DATA_BLOCK "ST10_DeviceError"
{ S7_Optimized_Access := 'FALSE' }
VERSION : 0.1
   STRUCT
      CylinderFault : Struct
         C1GoWorkFault : Bool;
         C1GoHomeFault : Bool;
         C1SensorPositionFault : Bool;
         C1SpareFault : Bool;
         C2GoWorkFault : Bool;
         C2GoHomeFault : Bool;
         C2SensorPositionFault : Bool;
         C2SpareFault : Bool;
         C3GoWorkFault : Bool;
         C3GoHomeFault : Bool;
         C3SensorPositionFault : Bool;
         C3SpareFault : Bool;
         C4GoWorkFault : Bool;
         C4GoHomeFault : Bool;
         C4SensorPositionFault : Bool;
         C4SpareFault : Bool;
         C5GoWorkFault : Bool;
         C5GoHomeFault : Bool;
         C5SensorPositionFault : Bool;
         C5SpareFault : Bool;
         C6GoWorkFault : Bool;
         C6GoHomeFault : Bool;
         C6SensorPositionFault : Bool;
         C6SpareFault : Bool;
         C7GoWorkFault : Bool;
         C7GoHomeFault : Bool;
         C7SensorPositionFault : Bool;
         C7SpareFault : Bool;
         C8GoWorkFault : Bool;
         C8GoHomeFault : Bool;
         C8SensorPositionFault : Bool;
         C8SpareFault : Bool;
         C9GoWorkFault : Bool;
         C9GoHomeFault : Bool;
         C9SensorPositionFault : Bool;
         C9SpareFault : Bool;
         C10GoWorkFault : Bool;
         C10GoHomeFault : Bool;
         C10SensorPositionFault : Bool;
         C10SpareFault : Bool;
         C11GoWorkFault : Bool;
         C11GoHomeFault : Bool;
         C11SensorPositionFault : Bool;
         C11SpareFault : Bool;
         C12GoWorkFault : Bool;
         C12GoHomeFault : Bool;
         C12SensorPositionFault : Bool;
         C12SpareFault : Bool;
         C13GoWorkFault : Bool;
         C13GoHomeFault : Bool;
         C13SensorPositionFault : Bool;
         C13SpareFault : Bool;
         C14GoWorkFault : Bool;
         C14GoHomeFault : Bool;
         C14SensorPositionFault : Bool;
         C14SpareFault : Bool;
         C15GoWorkFault : Bool;
         C15GoHomeFault : Bool;
         C15SensorPositionFault : Bool;
         C15SpareFault : Bool;
         C16GoWorkFault : Bool;
         C16GoHomeFault : Bool;
         C16SensorPositionFault : Bool;
         C16SpareFault : Bool;
         C17GoWorkFault : Bool;
         C17GoHomeFault : Bool;
         C17SensorPositionFault : Bool;
         C17SpareFault : Bool;
         C18GoWorkFault : Bool;
         C18GoHomeFault : Bool;
         C18SensorPositionFault : Bool;
         C18SpareFault : Bool;
         C19GoWorkFault : Bool;
         C19GoHomeFault : Bool;
         C19SensorPositionFault : Bool;
         C19SpareFault : Bool;
         C20GoWorkFault : Bool;
         C20GoHomeFault : Bool;
         C20SensorPositionFault : Bool;
         C20SpareFault : Bool;
         C21GoWorkFault : Bool;
         C21GoHomeFault : Bool;
         C21SensorPositionFault : Bool;
         C21SpareFault : Bool;
         C22GoWorkFault : Bool;
         C22GoHomeFault : Bool;
         C22SensorPositionFault : Bool;
         C22SpareFault : Bool;
         C23GoWorkFault : Bool;
         C23GoHomeFault : Bool;
         C23SensorPositionFault : Bool;
         C23SpareFault : Bool;
         C24GoWorkFault : Bool;
         C24GoHomeFault : Bool;
         C24SensorPositionFault : Bool;
         C24SpareFault : Bool;
         C25GoWorkFault : Bool;
         C25GoHomeFault : Bool;
         C25SensorPositionFault : Bool;
         C25SpareFault : Bool;
         C26GoWorkFault : Bool;
         C26GoHomeFault : Bool;
         C26SensorPositionFault : Bool;
         C26SpareFault : Bool;
         C27GoWorkFault : Bool;
         C27GoHomeFault : Bool;
         C27SensorPositionFault : Bool;
         C27SpareFault : Bool;
         C28GoWorkFault : Bool;
         C28GoHomeFault : Bool;
         C28SensorPositionFault : Bool;
         C28SpareFault : Bool;
         C29GoWorkFault : Bool;
         C29GoHomeFault : Bool;
         C29SensorPositionFault : Bool;
         C29SpareFault : Bool;
         C30GoWorkFault : Bool;
         C30GoHomeFault : Bool;
         C30SensorPositionFault : Bool;
         C30SpareFault : Bool;
         C31GoWorkFault : Bool;
         C31GoHomeFault : Bool;
         C31SensorPositionFault : Bool;
         C31SpareFault : Bool;
         C32GoWorkFault : Bool;
         C32GoHomeFault : Bool;
         C32SensorPositionFault : Bool;
         C32SpareFault : Bool;
         C33GoWorkFault : Bool;
         C33GoHomeFault : Bool;
         C33SensorPositionFault : Bool;
         C33SpareFault : Bool;
         C34GoWorkFault : Bool;
         C34GoHomeFault : Bool;
         C34SensorPositionFault : Bool;
         C34SpareFault : Bool;
         C35GoWorkFault : Bool;
         C35GoHomeFault : Bool;
         C35SensorPositionFault : Bool;
         C35SpareFault : Bool;
         C36GoWorkFault : Bool;
         C36GoHomeFault : Bool;
         C36SensorPositionFault : Bool;
         C36SpareFault : Bool;
         C37GoWorkFault : Bool;
         C37GoHomeFault : Bool;
         C37SensorPositionFault : Bool;
         C37SpareFault : Bool;
         C38GoWorkFault : Bool;
         C38GoHomeFault : Bool;
         C38SensorPositionFault : Bool;
         C38SpareFault : Bool;
         C39GoWorkFault : Bool;
         C39GoHomeFault : Bool;
         C39SensorPositionFault : Bool;
         C39SpareFault : Bool;
         C40GoWorkFault : Bool;
         C40GoHomeFault : Bool;
         C40SensorPositionFault : Bool;
         C40SpareFault : Bool;
         C41GoWorkFault : Bool;
         C41GoHomeFault : Bool;
         C41SensorPositionFault : Bool;
         C41SpareFault : Bool;
         C42GoWorkFault : Bool;
         C42GoHomeFault : Bool;
         C42SensorPositionFault : Bool;
         C42SpareFault : Bool;
         C43GoWorkFault : Bool;
         C43GoHomeFault : Bool;
         C43SensorPositionFault : Bool;
         C43SpareFault : Bool;
         C44GoWorkFault : Bool;
         C44GoHomeFault : Bool;
         C44SensorPositionFault : Bool;
         C44SpareFault : Bool;
         C45GoWorkFault : Bool;
         C45GoHomeFault : Bool;
         C45SensorPositionFault : Bool;
         C45SpareFault : Bool;
         C46GoWorkFault : Bool;
         C46GoHomeFault : Bool;
         C46SensorPositionFault : Bool;
         C46SpareFault : Bool;
         C47GoWorkFault : Bool;
         C47GoHomeFault : Bool;
         C47SensorPositionFault : Bool;
         C47SpareFault : Bool;
         C48GoWorkFault : Bool;
         C48GoHomeFault : Bool;
         C48SensorPositionFault : Bool;
         C48SpareFault : Bool;
         C49GoWorkFault : Bool;
         C49GoHomeFault : Bool;
         C49SensorPositionFault : Bool;
         C49SpareFault : Bool;
         C50GoWorkFault : Bool;
         C50GoHomeFault : Bool;
         C50SensorPositionFault : Bool;
         C50SpareFault : Bool;
         C51GoWorkFault : Bool;
         C51GoHomeFault : Bool;
         C51SensorPositionFault : Bool;
         C51SpareFault : Bool;
         C52GoWorkFault : Bool;
         C52GoHomeFault : Bool;
         C52SensorPositionFault : Bool;
         C52SpareFault : Bool;
         C53GoWorkFault : Bool;
         C53GoHomeFault : Bool;
         C53SensorPositionFault : Bool;
         C53SpareFault : Bool;
         C54GoWorkFault : Bool;
         C54GoHomeFault : Bool;
         C54SensorPositionFault : Bool;
         C54SpareFault : Bool;
         C55GoWorkFault : Bool;
         C55GoHomeFault : Bool;
         C55SensorPositionFault : Bool;
         C55SpareFault : Bool;
         C56GoWorkFault : Bool;
         C56GoHomeFault : Bool;
         C56SensorPositionFault : Bool;
         C56SpareFault : Bool;
         C57GoWorkFault : Bool;
         C57GoHomeFault : Bool;
         C57SensorPositionFault : Bool;
         C57SpareFault : Bool;
         C58GoWorkFault : Bool;
         C58GoHomeFault : Bool;
         C58SensorPositionFault : Bool;
         C58SpareFault : Bool;
         C59GoWorkFault : Bool;
         C59GoHomeFault : Bool;
         C59SensorPositionFault : Bool;
         C59SpareFault : Bool;
         C60GoWorkFault : Bool;
         C60GoHomeFault : Bool;
         C60SensorPositionFault : Bool;
         C60SpareFault : Bool;
         C61GoWorkFault : Bool;
         C61GoHomeFault : Bool;
         C61SensorPositionFault : Bool;
         C61SpareFault : Bool;
         C62GoWorkFault : Bool;
         C62GoHomeFault : Bool;
         C62SensorPositionFault : Bool;
         C62SpareFault : Bool;
         C63GoWorkFault : Bool;
         C63GoHomeFault : Bool;
         C63SensorPositionFault : Bool;
         C63SpareFault : Bool;
         C64GoWorkFault : Bool;
         C64GoHomeFault : Bool;
         C64SensorPositionFault : Bool;
         C64SpareFault : Bool;
         C65GoWorkFault : Bool;
         C65GoHomeFault : Bool;
         C65SensorPositionFault : Bool;
         C65SpareFault : Bool;
         C66GoWorkFault : Bool;
         C66GoHomeFault : Bool;
         C66SensorPositionFault : Bool;
         C66SpareFault : Bool;
         C67GoWorkFault : Bool;
         C67GoHomeFault : Bool;
         C67SensorPositionFault : Bool;
         C67SpareFault : Bool;
         C68GoWorkFault : Bool;
         C68GoHomeFault : Bool;
         C68SensorPositionFault : Bool;
         C68SpareFault : Bool;
         C69GoWorkFault : Bool;
         C69GoHomeFault : Bool;
         C69SensorPositionFault : Bool;
         C69SpareFault : Bool;
         C70GoWorkFault : Bool;
         C70GoHomeFault : Bool;
         C70SensorPositionFault : Bool;
         C70SpareFault : Bool;
         C71GoWorkFault : Bool;
         C71GoHomeFault : Bool;
         C71SensorPositionFault : Bool;
         C71SpareFault : Bool;
         C72GoWorkFault : Bool;
         C72GoHomeFault : Bool;
         C72SensorPositionFault : Bool;
         C72SpareFault : Bool;
         C73GoWorkFault : Bool;
         C73GoHomeFault : Bool;
         C73SensorPositionFault : Bool;
         C73SpareFault : Bool;
         C74GoWorkFault : Bool;
         C74GoHomeFault : Bool;
         C74SensorPositionFault : Bool;
         C74SpareFault : Bool;
         C75GoWorkFault : Bool;
         C75GoHomeFault : Bool;
         C75SensorPositionFault : Bool;
         C75SpareFault : Bool;
         C76GoWorkFault : Bool;
         C76GoHomeFault : Bool;
         C76SensorPositionFault : Bool;
         C76SpareFault : Bool;
         C77GoWorkFault : Bool;
         C77GoHomeFault : Bool;
         C77SensorPositionFault : Bool;
         C77SpareFault : Bool;
         C78GoWorkFault : Bool;
         C78GoHomeFault : Bool;
         C78SensorPositionFault : Bool;
         C78SpareFault : Bool;
         C79GoWorkFault : Bool;
         C79GoHomeFault : Bool;
         C79SensorPositionFault : Bool;
         C79SpareFault : Bool;
         C80GoWorkFault : Bool;
         C80GoHomeFault : Bool;
         C80SensorPositionFault : Bool;
         C80SpareFault : Bool;
         C81GoWorkFault : Bool;
         C81GoHomeFault : Bool;
         C81SensorPositionFault : Bool;
         C81SpareFault : Bool;
         C82GoWorkFault : Bool;
         C82GoHomeFault : Bool;
         C82SensorPositionFault : Bool;
         C82SpareFault : Bool;
         C83GoWorkFault : Bool;
         C83GoHomeFault : Bool;
         C83SensorPositionFault : Bool;
         C83SpareFault : Bool;
         C84GoWorkFault : Bool;
         C84GoHomeFault : Bool;
         C84SensorPositionFault : Bool;
         C84SpareFault : Bool;
         C85GoWorkFault : Bool;
         C85GoHomeFault : Bool;
         C85SensorPositionFault : Bool;
         C85SpareFault : Bool;
         C86GoWorkFault : Bool;
         C86GoHomeFault : Bool;
         C86SensorPositionFault : Bool;
         C86SpareFault : Bool;
         C87GoWorkFault : Bool;
         C87GoHomeFault : Bool;
         C87SensorPositionFault : Bool;
         C87SpareFault : Bool;
         C88GoWorkFault : Bool;
         C88GoHomeFault : Bool;
         C88SensorPositionFault : Bool;
         C88SpareFault : Bool;
         C89GoWorkFault : Bool;
         C89GoHomeFault : Bool;
         C89SensorPositionFault : Bool;
         C89SpareFault : Bool;
         C90GoWorkFault : Bool;
         C90GoHomeFault : Bool;
         C90SensorPositionFault : Bool;
         C90SpareFault : Bool;
         C91GoWorkFault : Bool;
         C91GoHomeFault : Bool;
         C91SensorPositionFault : Bool;
         C91SpareFault : Bool;
         C92GoWorkFault : Bool;
         C92GoHomeFault : Bool;
         C92SensorPositionFault : Bool;
         C92SpareFault : Bool;
         C93GoWorkFault : Bool;
         C93GoHomeFault : Bool;
         C93SensorPositionFault : Bool;
         C93SpareFault : Bool;
         C94GoWorkFault : Bool;
         C94GoHomeFault : Bool;
         C94SensorPositionFault : Bool;
         C94SpareFault : Bool;
         C95GoWorkFault : Bool;
         C95GoHomeFault : Bool;
         C95SensorPositionFault : Bool;
         C95SpareFault : Bool;
         C96GoWorkFault : Bool;
         C96GoHomeFault : Bool;
         C96SensorPositionFault : Bool;
         C96SpareFault : Bool;
         C97GoWorkFault : Bool;
         C97GoHomeFault : Bool;
         C97SensorPositionFault : Bool;
         C97SpareFault : Bool;
         C98GoWorkFault : Bool;
         C98GoHomeFault : Bool;
         C98SensorPositionFault : Bool;
         C98SpareFault : Bool;
         C99GoWorkFault : Bool;
         C99GoHomeFault : Bool;
         C99SensorPositionFault : Bool;
         C99SpareFault : Bool;
         C100GoWorkFault : Bool;
         C100GoHomeFault : Bool;
         C100SensorPositionFault : Bool;
         C100SpareFault : Bool;
         C101GoWorkFault : Bool;
         C101GoHomeFault : Bool;
         C101SensorPositionFault : Bool;
         C101SpareFault : Bool;
         C102GoWorkFault : Bool;
         C102GoHomeFault : Bool;
         C102SensorPositionFault : Bool;
         C102SpareFault : Bool;
         C103GoWorkFault : Bool;
         C103GoHomeFault : Bool;
         C103SensorPositionFault : Bool;
         C103SpareFault : Bool;
         C104GoWorkFault : Bool;
         C104GoHomeFault : Bool;
         C104SensorPositionFault : Bool;
         C104SpareFault : Bool;
         C105GoWorkFault : Bool;
         C105GoHomeFault : Bool;
         C105SensorPositionFault : Bool;
         C105SpareFault : Bool;
         C106GoWorkFault : Bool;
         C106GoHomeFault : Bool;
         C106SensorPositionFault : Bool;
         C106SpareFault : Bool;
         C107GoWorkFault : Bool;
         C107GoHomeFault : Bool;
         C107SensorPositionFault : Bool;
         C107SpareFault : Bool;
         C108GoWorkFault : Bool;
         C108GoHomeFault : Bool;
         C108SensorPositionFault : Bool;
         C108SpareFault : Bool;
         C109GoWorkFault : Bool;
         C109GoHomeFault : Bool;
         C109SensorPositionFault : Bool;
         C109SpareFault : Bool;
         C110GoWorkFault : Bool;
         C110GoHomeFault : Bool;
         C110SensorPositionFault : Bool;
         C110SpareFault : Bool;
         C111GoWorkFault : Bool;
         C111GoHomeFault : Bool;
         C111SensorPositionFault : Bool;
         C111SpareFault : Bool;
         C112GoWorkFault : Bool;
         C112GoHomeFault : Bool;
         C112SensorPositionFault : Bool;
         C112SpareFault : Bool;
         C113GoWorkFault : Bool;
         C113GoHomeFault : Bool;
         C113SensorPositionFault : Bool;
         C113SpareFault : Bool;
         C114GoWorkFault : Bool;
         C114GoHomeFault : Bool;
         C114SensorPositionFault : Bool;
         C114SpareFault : Bool;
         C115GoWorkFault : Bool;
         C115GoHomeFault : Bool;
         C115SensorPositionFault : Bool;
         C115SpareFault : Bool;
         C116GoWorkFault : Bool;
         C116GoHomeFault : Bool;
         C116SensorPositionFault : Bool;
         C116SpareFault : Bool;
         C117GoWorkFault : Bool;
         C117GoHomeFault : Bool;
         C117SensorPositionFault : Bool;
         C117SpareFault : Bool;
         C118GoWorkFault : Bool;
         C118GoHomeFault : Bool;
         C118SensorPositionFault : Bool;
         C118SpareFault : Bool;
         C119GoWorkFault : Bool;
         C119GoHomeFault : Bool;
         C119SensorPositionFault : Bool;
         C119SpareFault : Bool;
         C120GoWorkFault : Bool;
         C120GoHomeFault : Bool;
         C120SensorPositionFault : Bool;
         C120SpareFault : Bool;
         C121GoWorkFault : Bool;
         C121GoHomeFault : Bool;
         C121SensorPositionFault : Bool;
         C121SpareFault : Bool;
         C122GoWorkFault : Bool;
         C122GoHomeFault : Bool;
         C122SensorPositionFault : Bool;
         C122SpareFault : Bool;
         C123GoWorkFault : Bool;
         C123GoHomeFault : Bool;
         C123SensorPositionFault : Bool;
         C123SpareFault : Bool;
         C124GoWorkFault : Bool;
         C124GoHomeFault : Bool;
         C124SensorPositionFault : Bool;
         C124SpareFault : Bool;
         C125GoWorkFault : Bool;
         C125GoHomeFault : Bool;
         C125SensorPositionFault : Bool;
         C125SpareFault : Bool;
         C126GoWorkFault : Bool;
         C126GoHomeFault : Bool;
         C126SensorPositionFault : Bool;
         C126SpareFault : Bool;
         C127GoWorkFault : Bool;
         C127GoHomeFault : Bool;
         C127SensorPositionFault : Bool;
         C127SpareFault : Bool;
         C128GoWorkFault : Bool;
         C128GoHomeFault : Bool;
         C128SensorPositionFault : Bool;
         C128SpareFault : Bool;
         C129GoWorkFault : Bool;
         C129GoHomeFault : Bool;
         C129SensorPositionFault : Bool;
         C129SpareFault : Bool;
         C130GoWorkFault : Bool;
         C130GoHomeFault : Bool;
         C130SensorPositionFault : Bool;
         C130SpareFault : Bool;
         C131GoWorkFault : Bool;
         C131GoHomeFault : Bool;
         C131SensorPositionFault : Bool;
         C131SpareFault : Bool;
         C132GoWorkFault : Bool;
         C132GoHomeFault : Bool;
         C132SensorPositionFault : Bool;
         C132SpareFault : Bool;
         C133GoWorkFault : Bool;
         C133GoHomeFault : Bool;
         C133SensorPositionFault : Bool;
         C133SpareFault : Bool;
         C134GoWorkFault : Bool;
         C134GoHomeFault : Bool;
         C134SensorPositionFault : Bool;
         C134SpareFault : Bool;
         C135GoWorkFault : Bool;
         C135GoHomeFault : Bool;
         C135SensorPositionFault : Bool;
         C135SpareFault : Bool;
         C136GoWorkFault : Bool;
         C136GoHomeFault : Bool;
         C136SensorPositionFault : Bool;
         C136SpareFault : Bool;
         C137GoWorkFault : Bool;
         C137GoHomeFault : Bool;
         C137SensorPositionFault : Bool;
         C137SpareFault : Bool;
         C138GoWorkFault : Bool;
         C138GoHomeFault : Bool;
         C138SensorPositionFault : Bool;
         C138SpareFault : Bool;
         C139GoWorkFault : Bool;
         C139GoHomeFault : Bool;
         C139SensorPositionFault : Bool;
         C139SpareFault : Bool;
         C140GoWorkFault : Bool;
         C140GoHomeFault : Bool;
         C140SensorPositionFault : Bool;
         C140SpareFault : Bool;
         C141GoWorkFault : Bool;
         C141GoHomeFault : Bool;
         C141SensorPositionFault : Bool;
         C141SpareFault : Bool;
         C142GoWorkFault : Bool;
         C142GoHomeFault : Bool;
         C142SensorPositionFault : Bool;
         C142SpareFault : Bool;
         C143GoWorkFault : Bool;
         C143GoHomeFault : Bool;
         C143SensorPositionFault : Bool;
         C143SpareFault : Bool;
         C144GoWorkFault : Bool;
         C144GoHomeFault : Bool;
         C144SensorPositionFault : Bool;
         C144SpareFault : Bool;
         C145GoWorkFault : Bool;
         C145GoHomeFault : Bool;
         C145SensorPositionFault : Bool;
         C145SpareFault : Bool;
         C146GoWorkFault : Bool;
         C146GoHomeFault : Bool;
         C146SensorPositionFault : Bool;
         C146SpareFault : Bool;
         C147GoWorkFault : Bool;
         C147GoHomeFault : Bool;
         C147SensorPositionFault : Bool;
         C147SpareFault : Bool;
         C148GoWorkFault : Bool;
         C148GoHomeFault : Bool;
         C148SensorPositionFault : Bool;
         C148SpareFault : Bool;
         C149GoWorkFault : Bool;
         C149GoHomeFault : Bool;
         C149SensorPositionFault : Bool;
         C149SpareFault : Bool;
         C150GoWorkFault : Bool;
         C150GoHomeFault : Bool;
         C150SensorPositionFault : Bool;
         C150SpareFault : Bool;
         C151GoWorkFault : Bool;
         C151GoHomeFault : Bool;
         C151SensorPositionFault : Bool;
         C151SpareFault : Bool;
         C152GoWorkFault : Bool;
         C152GoHomeFault : Bool;
         C152SensorPositionFault : Bool;
         C152SpareFault : Bool;
         C153GoWorkFault : Bool;
         C153GoHomeFault : Bool;
         C153SensorPositionFault : Bool;
         C153SpareFault : Bool;
         C154GoWorkFault : Bool;
         C154GoHomeFault : Bool;
         C154SensorPositionFault : Bool;
         C154SpareFault : Bool;
         C155GoWorkFault : Bool;
         C155GoHomeFault : Bool;
         C155SensorPositionFault : Bool;
         C155SpareFault : Bool;
         C156GoWorkFault : Bool;
         C156GoHomeFault : Bool;
         C156SensorPositionFault : Bool;
         C156SpareFault : Bool;
         C157GoWorkFault : Bool;
         C157GoHomeFault : Bool;
         C157SensorPositionFault : Bool;
         C157SpareFault : Bool;
         C158GoWorkFault : Bool;
         C158GoHomeFault : Bool;
         C158SensorPositionFault : Bool;
         C158SpareFault : Bool;
         C159GoWorkFault : Bool;
         C159GoHomeFault : Bool;
         C159SensorPositionFault : Bool;
         C159SpareFault : Bool;
         C160GoWorkFault : Bool;
         C160GoHomeFault : Bool;
         C160SensorPositionFault : Bool;
         C160SpareFault : Bool;
         C161GoWorkFault : Bool;
         C161GoHomeFault : Bool;
         C161SensorPositionFault : Bool;
         C161SpareFault : Bool;
         C162GoWorkFault : Bool;
         C162GoHomeFault : Bool;
         C162SensorPositionFault : Bool;
         C162SpareFault : Bool;
         C163GoWorkFault : Bool;
         C163GoHomeFault : Bool;
         C163SensorPositionFault : Bool;
         C163SpareFault : Bool;
         C164GoWorkFault : Bool;
         C164GoHomeFault : Bool;
         C164SensorPositionFault : Bool;
         C164SpareFault : Bool;
         C165GoWorkFault : Bool;
         C165GoHomeFault : Bool;
         C165SensorPositionFault : Bool;
         C165SpareFault : Bool;
         C166GoWorkFault : Bool;
         C166GoHomeFault : Bool;
         C166SensorPositionFault : Bool;
         C166SpareFault : Bool;
         C167GoWorkFault : Bool;
         C167GoHomeFault : Bool;
         C167SensorPositionFault : Bool;
         C167SpareFault : Bool;
         C168GoWorkFault : Bool;
         C168GoHomeFault : Bool;
         C168SensorPositionFault : Bool;
         C168SpareFault : Bool;
         C169GoWorkFault : Bool;
         C169GoHomeFault : Bool;
         C169SensorPositionFault : Bool;
         C169SpareFault : Bool;
         C170GoWorkFault : Bool;
         C170GoHomeFault : Bool;
         C170SensorPositionFault : Bool;
         C170SpareFault : Bool;
         C171GoWorkFault : Bool;
         C171GoHomeFault : Bool;
         C171SensorPositionFault : Bool;
         C171SpareFault : Bool;
         C172GoWorkFault : Bool;
         C172GoHomeFault : Bool;
         C172SensorPositionFault : Bool;
         C172SpareFault : Bool;
         C173GoWorkFault : Bool;
         C173GoHomeFault : Bool;
         C173SensorPositionFault : Bool;
         C173SpareFault : Bool;
         C174GoWorkFault : Bool;
         C174GoHomeFault : Bool;
         C174SensorPositionFault : Bool;
         C174SpareFault : Bool;
         C175GoWorkFault : Bool;
         C175GoHomeFault : Bool;
         C175SensorPositionFault : Bool;
         C175SpareFault : Bool;
         C176GoWorkFault : Bool;
         C176GoHomeFault : Bool;
         C176SensorPositionFault : Bool;
         C176SpareFault : Bool;
         C177GoWorkFault : Bool;
         C177GoHomeFault : Bool;
         C177SensorPositionFault : Bool;
         C177SpareFault : Bool;
         C178GoWorkFault : Bool;
         C178GoHomeFault : Bool;
         C178SensorPositionFault : Bool;
         C178SpareFault : Bool;
         C179GoWorkFault : Bool;
         C179GoHomeFault : Bool;
         C179SensorPositionFault : Bool;
         C179SpareFault : Bool;
         C180GoWorkFault : Bool;
         C180GoHomeFault : Bool;
         C180SensorPositionFault : Bool;
         C180SpareFault : Bool;
         C181GoWorkFault : Bool;
         C181GoHomeFault : Bool;
         C181SensorPositionFault : Bool;
         C181SpareFault : Bool;
         C182GoWorkFault : Bool;
         C182GoHomeFault : Bool;
         C182SensorPositionFault : Bool;
         C182SpareFault : Bool;
         C183GoWorkFault : Bool;
         C183GoHomeFault : Bool;
         C183SensorPositionFault : Bool;
         C183SpareFault : Bool;
         C184GoWorkFault : Bool;
         C184GoHomeFault : Bool;
         C184SensorPositionFault : Bool;
         C184SpareFault : Bool;
         C185GoWorkFault : Bool;
         C185GoHomeFault : Bool;
         C185SensorPositionFault : Bool;
         C185SpareFault : Bool;
         C186GoWorkFault : Bool;
         C186GoHomeFault : Bool;
         C186SensorPositionFault : Bool;
         C186SpareFault : Bool;
         C187GoWorkFault : Bool;
         C187GoHomeFault : Bool;
         C187SensorPositionFault : Bool;
         C187SpareFault : Bool;
         C188GoWorkFault : Bool;
         C188GoHomeFault : Bool;
         C188SensorPositionFault : Bool;
         C188SpareFault : Bool;
         C189GoWorkFault : Bool;
         C189GoHomeFault : Bool;
         C189SensorPositionFault : Bool;
         C189SpareFault : Bool;
         C190GoWorkFault : Bool;
         C190GoHomeFault : Bool;
         C190SensorPositionFault : Bool;
         C190SpareFault : Bool;
         C191GoWorkFault : Bool;
         C191GoHomeFault : Bool;
         C191SensorPositionFault : Bool;
         C191SpareFault : Bool;
         C192GoWorkFault : Bool;
         C192GoHomeFault : Bool;
         C192SensorPositionFault : Bool;
         C192SpareFault : Bool;
         C193GoWorkFault : Bool;
         C193GoHomeFault : Bool;
         C193SensorPositionFault : Bool;
         C193SpareFault : Bool;
         C194GoWorkFault : Bool;
         C194GoHomeFault : Bool;
         C194SensorPositionFault : Bool;
         C194SpareFault : Bool;
         C195GoWorkFault : Bool;
         C195GoHomeFault : Bool;
         C195SensorPositionFault : Bool;
         C195SpareFault : Bool;
         C196GoWorkFault : Bool;
         C196GoHomeFault : Bool;
         C196SensorPositionFault : Bool;
         C196SpareFault : Bool;
         C197GoWorkFault : Bool;
         C197GoHomeFault : Bool;
         C197SensorPositionFault : Bool;
         C197SpareFault : Bool;
         C198GoWorkFault : Bool;
         C198GoHomeFault : Bool;
         C198SensorPositionFault : Bool;
         C198SpareFault : Bool;
         C199GoWorkFault : Bool;
         C199GoHomeFault : Bool;
         C199SensorPositionFault : Bool;
         C199SpareFault : Bool;
         C200GoWorkFault : Bool;
         C200GoHomeFault : Bool;
         C200SensorPositionFault : Bool;
         C200SpareFault : Bool;
      END_STRUCT;
      A : Struct
         A1TableScan : Struct
            LightCuritTouch : Bool;
            ScanCodeNG : Bool;
            "3" : Bool;
            "4" : Bool;
            "5" : Bool;
            "6" : Bool;
            "7" : Bool;
            "8" : Bool;
            "9" : Bool;
            "10" : Bool;
            "11" : Bool;
            "12" : Bool;
            "13" : Bool;
            "14" : Bool;
            "15" : Bool;
            "16" : Bool;
         END_STRUCT;
         A1TableUnloading : Struct
            LackMaterial : Bool;
            RingCheckExist : Bool;
            "3" : Bool;
            "4" : Bool;
            "5" : Bool;
            "6" : Bool;
            "7" : Bool;
            "8" : Bool;
            "9" : Bool;
            "10" : Bool;
            "11" : Bool;
            "12" : Bool;
            "13" : Bool;
            "14" : Bool;
            "15" : Bool;
            "16" : Bool;
         END_STRUCT;
         A1RotaryScan : Struct
            ProductAnomaly : Bool;
            PartMissing : Bool;
            "3" : Bool;
            "4" : Bool;
            "5" : Bool;
            "6" : Bool;
            "7" : Bool;
            "8" : Bool;
            "9" : Bool;
            "10" : Bool;
            "11" : Bool;
            "12" : Bool;
            "13" : Bool;
            "14" : Bool;
            "15" : Bool;
            "16" : Bool;
         END_STRUCT;
         A1FixtureCodeScan : Struct
            ReadNG_1 : Bool;
            ReadNG_2 : Bool;
            ReadNG_3 : Bool;
            ReadNG_4 : Bool;
            ReadNG_5 : Bool;
            ReadNG_6 : Bool;
            ReadNG_7 : Bool;
            ReadNG_8 : Bool;
            ReadNG_9 : Bool;
            ReadNG_10 : Bool;
            ReadNG_11 : Bool;
            ReadNG_12 : Bool;
            ReadNG_13 : Bool;
            "14" : Bool;
            "15" : Bool;
            "16" : Bool;
         END_STRUCT;
         A2TableScan : Struct
            LightCuritTouch : Bool;
            ScanCodeNG : Bool;
            "3" : Bool;
            "4" : Bool;
            "5" : Bool;
            "6" : Bool;
            "7" : Bool;
            "8" : Bool;
            "9" : Bool;
            "10" : Bool;
            "11" : Bool;
            "12" : Bool;
            "13" : Bool;
            "14" : Bool;
            "15" : Bool;
            "16" : Bool;
         END_STRUCT;
         A2TableUnloading : Struct
            LackMaterial : Bool;
            RingCheckExist : Bool;
            "3" : Bool;
            "4" : Bool;
            "5" : Bool;
            "6" : Bool;
            "7" : Bool;
            "8" : Bool;
            "9" : Bool;
            "10" : Bool;
            "11" : Bool;
            "12" : Bool;
            "13" : Bool;
            "14" : Bool;
            "15" : Bool;
            "16" : Bool;
         END_STRUCT;
         A2RotaryScan : Struct
            "1" : Bool;
            "2" : Bool;
            "3" : Bool;
            "4" : Bool;
            "5" : Bool;
            "6" : Bool;
            "7" : Bool;
            "8" : Bool;
            "9" : Bool;
            "10" : Bool;
            "11" : Bool;
            "12" : Bool;
            "13" : Bool;
            "14" : Bool;
            "15" : Bool;
            "16" : Bool;
         END_STRUCT;
         A2FixtureCodeScan : Struct
            ReadNG_1 : Bool;
            ReadNG_2 : Bool;
            ReadNG_3 : Bool;
            ReadNG_4 : Bool;
            ReadNG_5 : Bool;
            ReadNG_6 : Bool;
            ReadNG_7 : Bool;
            ReadNG_8 : Bool;
            ReadNG_9 : Bool;
            ReadNG_10 : Bool;
            ReadNG_11 : Bool;
            ReadNG_12 : Bool;
            ReadNG_13 : Bool;
            "14" : Bool;
            "15" : Bool;
            "16" : Bool;
         END_STRUCT;
         Other : Struct
            Servo_380A1 : Bool;
            Servo_381A1 : Bool;
            Servo_383A1 : Bool;
            "4" : Bool;
            "5" : Bool;
            "6" : Bool;
            "7" : Bool;
            "8" : Bool;
            "9" : Bool;
            "10" : Bool;
            "11" : Bool;
            "12" : Bool;
            "13" : Bool;
            "14" : Bool;
            "15" : Bool;
            "16" : Bool;
         END_STRUCT;
         A_Spare_2 : Struct
            Servo_380A1 : Bool;
            Servo_381A1 : Bool;
            Scan_800A1 : Bool;
            Scan_801A1 : Bool;
            Scan_804A1 : Bool;
            "6" : Bool;
            "7" : Bool;
            "8" : Bool;
            "9" : Bool;
            "10" : Bool;
            "11" : Bool;
            "12" : Bool;
            "13" : Bool;
            "14" : Bool;
            "15" : Bool;
            "16" : Bool;
         END_STRUCT;
      END_STRUCT;
      B : Struct
         B1Press : Struct
            StatusError : Bool;
            ShaftSensorCheckError : Bool;
            RingSensorCheckError : Bool;
            "4" : Bool;
            "5" : Bool;
            "6" : Bool;
            "7" : Bool;
            "8" : Bool;
            "9" : Bool;
            "10" : Bool;
            "11" : Bool;
            "12" : Bool;
            "13" : Bool;
            "14" : Bool;
            "15" : Bool;
            "16" : Bool;
         END_STRUCT;
         B2Press : Struct
            StatusError : Bool;
            ShaftSensorCheckError : Bool;
            RingSensorCheckError : Bool;
            "4" : Bool;
            "5" : Bool;
            "6" : Bool;
            "7" : Bool;
            "8" : Bool;
            "9" : Bool;
            "10" : Bool;
            "11" : Bool;
            "12" : Bool;
            "13" : Bool;
            "14" : Bool;
            "15" : Bool;
            "16" : Bool;
         END_STRUCT;
         B_Spare_1 : Struct
            Kistler_Press1_372A1 : Bool;
            Scan_806A1 : Bool;
            Kistler_Press2_375A1 : Bool;
            "4" : Bool;
            "5" : Bool;
            "6" : Bool;
            "7" : Bool;
            "8" : Bool;
            "9" : Bool;
            "10" : Bool;
            "11" : Bool;
            "12" : Bool;
            "13" : Bool;
            "14" : Bool;
            "15" : Bool;
            "16" : Bool;
         END_STRUCT;
         B_Spare_2 : Struct
            "1" : Bool;
            "2" : Bool;
            "3" : Bool;
            "4" : Bool;
            "5" : Bool;
            "6" : Bool;
            "7" : Bool;
            "8" : Bool;
            "9" : Bool;
            "10" : Bool;
            "11" : Bool;
            "12" : Bool;
            "13" : Bool;
            "14" : Bool;
            "15" : Bool;
            "16" : Bool;
         END_STRUCT;
         B_Spare_3 : Struct
            "1" : Bool;
            "2" : Bool;
            "3" : Bool;
            "4" : Bool;
            "5" : Bool;
            "6" : Bool;
            "7" : Bool;
            "8" : Bool;
            "9" : Bool;
            "10" : Bool;
            "11" : Bool;
            "12" : Bool;
            "13" : Bool;
            "14" : Bool;
            "15" : Bool;
            "16" : Bool;
         END_STRUCT;
      END_STRUCT;
      C : Struct
         CGlueing : Struct
            SysError : Bool;
            StatusError : Bool;
            Servo_383A1 : Bool;
            Z : Bool;
            X : Bool;
            Y : Bool;
            "7" : Bool;
            "8" : Bool;
            "9" : Bool;
            "10" : Bool;
            "11" : Bool;
            "12" : Bool;
            "13" : Bool;
            "14" : Bool;
            "15" : Bool;
            "16" : Bool;
         END_STRUCT;
         Other : Struct
            Servo_383A1 : Bool;
            Z : Bool;
            X : Bool;
            Y : Bool;
            "5" : Bool;
            "6" : Bool;
            "7" : Bool;
            "8" : Bool;
            "9" : Bool;
            "10" : Bool;
            "11" : Bool;
            "12" : Bool;
            "13" : Bool;
            "14" : Bool;
            "15" : Bool;
            "16" : Bool;
         END_STRUCT;
         C_Spare_2 : Struct
            Servo_382A1 : Bool;
            IV3_810A1 : Bool;
            IV3_811A1 : Bool;
            GluingDeviceReady : Bool;
            GluingFault : Bool;
            GluingRefillTank : Bool;
            GluingTankEmpty : Bool;
            "8" : Bool;
            "9" : Bool;
            "10" : Bool;
            "11" : Bool;
            "12" : Bool;
            "13" : Bool;
            "14" : Bool;
            "15" : Bool;
            "16" : Bool;
         END_STRUCT;
         C_Spare_3 : Struct
            "1" : Bool;
            "2" : Bool;
            "3" : Bool;
            "4" : Bool;
            "5" : Bool;
            "6" : Bool;
            "7" : Bool;
            "8" : Bool;
            "9" : Bool;
            "10" : Bool;
            "11" : Bool;
            "12" : Bool;
            "13" : Bool;
            "14" : Bool;
            "15" : Bool;
            "16" : Bool;
         END_STRUCT;
         C_Spare_4 : Struct
            "1" : Bool;
            "2" : Bool;
            "3" : Bool;
            "4" : Bool;
            "5" : Bool;
            "6" : Bool;
            "7" : Bool;
            "8" : Bool;
            "9" : Bool;
            "10" : Bool;
            "11" : Bool;
            "12" : Bool;
            "13" : Bool;
            "14" : Bool;
            "15" : Bool;
            "16" : Bool;
         END_STRUCT;
      END_STRUCT;
      E : Struct
         NG_1 : Struct
            ShaftScanNGFull : Bool;
            PressNGFull : Bool;
            RingScanNGFull : Bool;
            ShaftScanStatus : Bool;
            PressNGStatus : Bool;
            RingScanNGStatus : Bool;
            "NG 1 DoorOpen" : Bool;
            "NG 2 DoorOpen" : Bool;
            "9" : Bool;
            "10" : Bool;
            "11" : Bool;
            "12" : Bool;
            "13" : Bool;
            "14" : Bool;
            "15" : Bool;
            "16" : Bool;
         END_STRUCT;
         NG_2 : Struct
            "Press/GlueNGFull" : Bool;
            MagnetNGFull : Bool;
            RingScanNGFull : Bool;
            "Press/GlueNGStatus" : Bool;
            MagnetNGStatus : Bool;
            RingScanNGStatus : Bool;
            "7" : Bool;
            "8" : Bool;
            "9" : Bool;
            "10" : Bool;
            "11" : Bool;
            "12" : Bool;
            "13" : Bool;
            "14" : Bool;
            "15" : Bool;
            "16" : Bool;
         END_STRUCT;
         E_Spare_1 : Struct
            "1" : Bool;
            "2" : Bool;
            "3" : Bool;
            "4" : Bool;
            "5" : Bool;
            "6" : Bool;
            "7" : Bool;
            "8" : Bool;
            "9" : Bool;
            "10" : Bool;
            "11" : Bool;
            "12" : Bool;
            "13" : Bool;
            "14" : Bool;
            "15" : Bool;
            "16" : Bool;
         END_STRUCT;
         E_Spare_2 : Struct
            "1" : Bool;
            "2" : Bool;
            "3" : Bool;
            "4" : Bool;
            "5" : Bool;
            "6" : Bool;
            "7" : Bool;
            "8" : Bool;
            "9" : Bool;
            "10" : Bool;
            "11" : Bool;
            "12" : Bool;
            "13" : Bool;
            "14" : Bool;
            "15" : Bool;
            "16" : Bool;
         END_STRUCT;
         E_Spare_3 : Struct
            "1" : Bool;
            "2" : Bool;
            "3" : Bool;
            "4" : Bool;
            "5" : Bool;
            "6" : Bool;
            "7" : Bool;
            "8" : Bool;
            "9" : Bool;
            "10" : Bool;
            "11" : Bool;
            "12" : Bool;
            "13" : Bool;
            "14" : Bool;
            "15" : Bool;
            "16" : Bool;
         END_STRUCT;
      END_STRUCT;
      F : Struct
         Robot_1 : Struct
            Grip1Error : Bool;
            Grip2Error : Bool;
            Grip1SensorCheckError : Bool;
            Grip2SensorCheckError : Bool;
            ManualMoved : Bool;
            "EXT Fault" : Bool;
            RobotNOTStart : Bool;
            "8" : Bool;
            "9" : Bool;
            "10" : Bool;
            "11" : Bool;
            "12" : Bool;
            "13" : Bool;
            "14" : Bool;
            "15" : Bool;
            "16" : Bool;
         END_STRUCT;
         Robot_2 : Struct
            Grip1Error : Bool;
            Grip2Error : Bool;
            Grip1SensorCheckError : Bool;
            Grip2SensorCheckError : Bool;
            ManualMoved : Bool;
            ReadNG_1 : Bool;
            ReadNG_2 : Bool;
            ReadNG_3 : Bool;
            ReadNG_4 : Bool;
            "EXT Fault" : Bool;
            RobotNOTStart : Bool;
            "12" : Bool;
            "13" : Bool;
            "14" : Bool;
            "15" : Bool;
            "16" : Bool;
         END_STRUCT;
         Robot_3 : Struct
            Grip1Error : Bool;
            Grip2Error : Bool;
            Grip1SensorCheckError : Bool;
            Grip2SensorCheckError : Bool;
            ManualMoved : Bool;
            "EXT Fault" : Bool;
            RobotNOTStart : Bool;
            "8" : Bool;
            "9" : Bool;
            "10" : Bool;
            "11" : Bool;
            "12" : Bool;
            "13" : Bool;
            "14" : Bool;
            "15" : Bool;
            "16" : Bool;
         END_STRUCT;
         F_Spare_1 : Struct
            Scan_805A1 : Bool;
            Robot_1 : Bool;
            Robot_2 : Bool;
            Robot_3 : Bool;
            "5" : Bool;
            "6" : Bool;
            "7" : Bool;
            "8" : Bool;
            "9" : Bool;
            "10" : Bool;
            "11" : Bool;
            "12" : Bool;
            "13" : Bool;
            "14" : Bool;
            "15" : Bool;
            "16" : Bool;
         END_STRUCT;
         F_Spare_2 : Struct
            "1" : Bool;
            "2" : Bool;
            "3" : Bool;
            "4" : Bool;
            "5" : Bool;
            "6" : Bool;
            "7" : Bool;
            "8" : Bool;
            "9" : Bool;
            "10" : Bool;
            "11" : Bool;
            "12" : Bool;
            "13" : Bool;
            "14" : Bool;
            "15" : Bool;
            "16" : Bool;
         END_STRUCT;
      END_STRUCT;
      H : Struct
         ShaftLine : Struct
            LiftingCylStatusError : Bool;
            LoadingStop1timeout : Bool;
            LoadingStop2timeout : Bool;
            LoadingStop3timeout : Bool;
            LoadingStop4timeout : Bool;
            UnloadingStop1timeout : Bool;
            UnloadingStop2timeout : Bool;
            UnloadingStop3timeout : Bool;
            UnloadingLiftingtimeout : Bool;
            EmptyStop1timeout : Bool;
            EmptyStop2timeout : Bool;
            EmptyStop3timeout : Bool;
            EmptyStop4timeout : Bool;
            "14" : Bool;
            "15" : Bool;
            "16" : Bool;
         END_STRUCT;
         Spare_1 : Struct
            "H-shaftLifting_Motor" : Bool;
            "H-shaftLoad_Motor" : Bool;
            "H-shaftUnLoad_Motor" : Bool;
            "4" : Bool;
            "5" : Bool;
            "6" : Bool;
            "7" : Bool;
            "8" : Bool;
            "9" : Bool;
            "10" : Bool;
            "11" : Bool;
            "12" : Bool;
            "13" : Bool;
            "14" : Bool;
            "15" : Bool;
            "16" : Bool;
         END_STRUCT;
         Spare_2 : Struct
            "1" : Bool;
            "2" : Bool;
            "3" : Bool;
            "4" : Bool;
            "5" : Bool;
            "6" : Bool;
            "7" : Bool;
            "8" : Bool;
            "9" : Bool;
            "10" : Bool;
            "11" : Bool;
            "12" : Bool;
            "13" : Bool;
            "14" : Bool;
            "15" : Bool;
            "16" : Bool;
         END_STRUCT;
         Spare_3 : Struct
            "1" : Bool;
            "2" : Bool;
            "3" : Bool;
            "4" : Bool;
            "5" : Bool;
            "6" : Bool;
            "7" : Bool;
            "8" : Bool;
            "9" : Bool;
            "10" : Bool;
            "11" : Bool;
            "12" : Bool;
            "13" : Bool;
            "14" : Bool;
            "15" : Bool;
            "16" : Bool;
         END_STRUCT;
         Spare_4 : Struct
            "1" : Bool;
            "2" : Bool;
            "3" : Bool;
            "4" : Bool;
            "5" : Bool;
            "6" : Bool;
            "7" : Bool;
            "8" : Bool;
            "9" : Bool;
            "10" : Bool;
            "11" : Bool;
            "12" : Bool;
            "13" : Bool;
            "14" : Bool;
            "15" : Bool;
            "16" : Bool;
         END_STRUCT;
      END_STRUCT;
      J : Struct
         MagnetLine : Struct
            LiftingCylStatusError : Bool;
            LoadingStop1timeout : Bool;
            LoadingStop2timeout : Bool;
            LoadingStop3timeout : Bool;
            LoadingStop4timeout : Bool;
            UnloadingStop1timeout : Bool;
            UnloadingStop2timeout : Bool;
            UnloadingStop3timeout : Bool;
            UnloadingLiftingtimeout : Bool;
            EmptyStop1timeout : Bool;
            EmptyStop2timeout : Bool;
            EmptyStop3timeout : Bool;
            EmptyStop4timeout : Bool;
            "14" : Bool;
            "15" : Bool;
            "16" : Bool;
         END_STRUCT;
         Spare_1 : Struct
            "J-MagnetLifting_Motor" : Bool;
            "J-MagnetLoad_Motor" : Bool;
            "J-MagnetUnLoad_Motor" : Bool;
            "4" : Bool;
            "5" : Bool;
            "6" : Bool;
            "7" : Bool;
            "8" : Bool;
            "9" : Bool;
            "10" : Bool;
            "11" : Bool;
            "12" : Bool;
            "13" : Bool;
            "14" : Bool;
            "15" : Bool;
            "16" : Bool;
         END_STRUCT;
         Spare_2 : Struct
            "1" : Bool;
            "2" : Bool;
            "3" : Bool;
            "4" : Bool;
            "5" : Bool;
            "6" : Bool;
            "7" : Bool;
            "8" : Bool;
            "9" : Bool;
            "10" : Bool;
            "11" : Bool;
            "12" : Bool;
            "13" : Bool;
            "14" : Bool;
            "15" : Bool;
            "16" : Bool;
         END_STRUCT;
         Spare_3 : Struct
            "1" : Bool;
            "2" : Bool;
            "3" : Bool;
            "4" : Bool;
            "5" : Bool;
            "6" : Bool;
            "7" : Bool;
            "8" : Bool;
            "9" : Bool;
            "10" : Bool;
            "11" : Bool;
            "12" : Bool;
            "13" : Bool;
            "14" : Bool;
            "15" : Bool;
            "16" : Bool;
         END_STRUCT;
         Spare_4 : Struct
            "1" : Bool;
            "2" : Bool;
            "3" : Bool;
            "4" : Bool;
            "5" : Bool;
            "6" : Bool;
            "7" : Bool;
            "8" : Bool;
            "9" : Bool;
            "10" : Bool;
            "11" : Bool;
            "12" : Bool;
            "13" : Bool;
            "14" : Bool;
            "15" : Bool;
            "16" : Bool;
         END_STRUCT;
      END_STRUCT;
      K : Struct
         ReserveLine : Struct
            LiftingCylStatusError : Bool;
            LoadingStop1timeout : Bool;
            LoadingStop2timeout : Bool;
            LoadingStop3timeout : Bool;
            LoadingStop4timeout : Bool;
            UnloadingStop1timeout : Bool;
            UnloadingStop2timeout : Bool;
            UnloadingStop3timeout : Bool;
            UnloadingLiftingtimeout : Bool;
            EmptyStop1timeout : Bool;
            EmptyStop2timeout : Bool;
            EmptyStop3timeout : Bool;
            EmptyStop4timeout : Bool;
            "14" : Bool;
            "15" : Bool;
            "16" : Bool;
         END_STRUCT;
         Spare_1 : Struct
            "K-Lifting_Motor" : Bool;
            "K-ReserveLoad_Motor" : Bool;
            "K-ReserveUnLoad_Motor" : Bool;
            "4" : Bool;
            "5" : Bool;
            "6" : Bool;
            "7" : Bool;
            "8" : Bool;
            "9" : Bool;
            "10" : Bool;
            "11" : Bool;
            "12" : Bool;
            "13" : Bool;
            "14" : Bool;
            "15" : Bool;
            "16" : Bool;
         END_STRUCT;
         Spare_2 : Struct
            "1" : Bool;
            "2" : Bool;
            "3" : Bool;
            "4" : Bool;
            "5" : Bool;
            "6" : Bool;
            "7" : Bool;
            "8" : Bool;
            "9" : Bool;
            "10" : Bool;
            "11" : Bool;
            "12" : Bool;
            "13" : Bool;
            "14" : Bool;
            "15" : Bool;
            "16" : Bool;
         END_STRUCT;
         Spare_3 : Struct
            "1" : Bool;
            "2" : Bool;
            "3" : Bool;
            "4" : Bool;
            "5" : Bool;
            "6" : Bool;
            "7" : Bool;
            "8" : Bool;
            "9" : Bool;
            "10" : Bool;
            "11" : Bool;
            "12" : Bool;
            "13" : Bool;
            "14" : Bool;
            "15" : Bool;
            "16" : Bool;
         END_STRUCT;
         Spare_4 : Struct
            "1" : Bool;
            "2" : Bool;
            "3" : Bool;
            "4" : Bool;
            "5" : Bool;
            "6" : Bool;
            "7" : Bool;
            "8" : Bool;
            "9" : Bool;
            "10" : Bool;
            "11" : Bool;
            "12" : Bool;
            "13" : Bool;
            "14" : Bool;
            "15" : Bool;
            "16" : Bool;
         END_STRUCT;
      END_STRUCT;
      L : Struct
         UnloadingLine : Struct
            UnloadingTransCylinderError : Bool;
            LoadingStop1timeout : Bool;
            LoadingStop2timeout : Bool;
            LoadingStop3timeout : Bool;
            LoadingStop4timeout : Bool;
            UnloadingStop1timeout : Bool;
            UnloadingStop2timeout : Bool;
            UnloadingStop3timeout : Bool;
            UnloadingLiftingtimeout : Bool;
            EmptyStop1timeout : Bool;
            EmptyStop2timeout : Bool;
            EmptyStop3timeout : Bool;
            EmptyStop4timeout : Bool;
            "14" : Bool;
            "15" : Bool;
            "16" : Bool;
         END_STRUCT;
         CuringOven : Struct
            "1" : Bool;
            "2" : Bool;
            "3" : Bool;
            "4" : Bool;
            "5" : Bool;
            "6" : Bool;
            "7" : Bool;
            "8" : Bool;
            "9" : Bool;
            "10" : Bool;
            "11" : Bool;
            "12" : Bool;
            "13" : Bool;
            "14" : Bool;
            "15" : Bool;
            "16" : Bool;
         END_STRUCT;
         Spare_2 : Struct
            "L-Unloading_Motor" : Bool;
            "L-Unloading _LineMotor" : Bool;
            "3" : Bool;
            "4" : Bool;
            "5" : Bool;
            "6" : Bool;
            "7" : Bool;
            "8" : Bool;
            "9" : Bool;
            "10" : Bool;
            "11" : Bool;
            "12" : Bool;
            "13" : Bool;
            "14" : Bool;
            "15" : Bool;
            "16" : Bool;
         END_STRUCT;
         Spare_3 : Struct
            "1" : Bool;
            "2" : Bool;
            "3" : Bool;
            "4" : Bool;
            "5" : Bool;
            "6" : Bool;
            "7" : Bool;
            "8" : Bool;
            "9" : Bool;
            "10" : Bool;
            "11" : Bool;
            "12" : Bool;
            "13" : Bool;
            "14" : Bool;
            "15" : Bool;
            "16" : Bool;
         END_STRUCT;
         Spare_4 : Struct
            "1" : Bool;
            "2" : Bool;
            "3" : Bool;
            "4" : Bool;
            "5" : Bool;
            "6" : Bool;
            "7" : Bool;
            "8" : Bool;
            "9" : Bool;
            "10" : Bool;
            "11" : Bool;
            "12" : Bool;
            "13" : Bool;
            "14" : Bool;
            "15" : Bool;
            "16" : Bool;
         END_STRUCT;
      END_STRUCT;
      MES_Error : Struct
         Offline : Bool;
         Reserved1_8 : Bool;
         CheckInCompOverTime_1 : Bool;
         CheckInResultOverTime_1 : Bool;
         CheckInCompOverTime_2 : Bool;
         CheckInResultOverTime_2 : Bool;
         CheckInCompOverTime_3 : Bool;
         CheckInResultOverTime_3 : Bool;
         CheckInCompOverTime_4 : Bool;
         CheckInResultOverTime_4 : Bool;
         CheckInCompOverTime_5 : Bool;
         CheckInResultOverTime_5 : Bool;
         CheckInCompOverTime_6 : Bool;
         CheckInResultOverTime_6 : Bool;
         CheckInCompOverTime_7 : Bool;
         CheckInResultOverTime_7 : Bool;
         CheckInCompOverTime_8 : Bool;
         CheckInResultOverTime_8 : Bool;
         CheckoutSaveResultNG : Bool;
         CheckoutCompRstOverTime : Bool;
         Reserved2_5 : Bool;
         Reserved2_6 : Bool;
         Reserved2_7 : Bool;
         SubCheck_CompOverTime : Bool;
         SubCheck_ResultOverTime : Bool;
         SubCheck_TriggerError : Bool;
         SubCheck_CheckResultNG : Bool;
         SubCheck_CompRstOverTime : Bool;
         Reserved3_5 : Bool;
         Reserved3_6 : Bool;
         Reserved3_7 : Bool;
         Processing_CompOverTime : Bool;
         Reserved4_1 : Bool;
         Processing_TriggerError : Bool;
         Reserved4_3 : Bool;
         Processing_CompRstOverTime : Bool;
         Reserved4_5 : Bool;
         Reserved4_6 : Bool;
         Reserved4_7 : Bool;
         Reserved5_0 : Bool;
         Reserved5_1 : Bool;
         Reserved5_2 : Bool;
         Reserved5_3 : Bool;
         Reserved5_4 : Bool;
         Reserved5_5 : Bool;
         Reserved5_6 : Bool;
         Reserved5_7 : Bool;
      END_STRUCT;
   END_STRUCT;


BEGIN

END_DATA_BLOCK

